Fanuc KAREL source: ka00001.KL

-- PROVISIONAL review KL for V1013-1; original PC SHA256 2018445ef6fb0ff1de9b7fd742bdcd096b2f0fa9a6b30116b0d319b35435d8ea
-- Incomplete behavior may be omitted. Consult companion uncertainty JSON. Do not deploy.
PROGRAM KA00001
%NOLOCKGROUP
VAR
  SRC : INTEGER
  DST : INTEGER
BEGIN
  -- UNRESOLVED_PC offsets 5-16; opcodes 2E,23
  -- UNRESOLVED_PC offsets 21-33; opcodes 21,23
  -- UNRESOLVED_PC offsets 38-42; opcodes 7F
END KA00001
